// Mitsubishi GX Works2 project: 供料   PLC: FX3U/FX3UC

PROGRAM MAIN
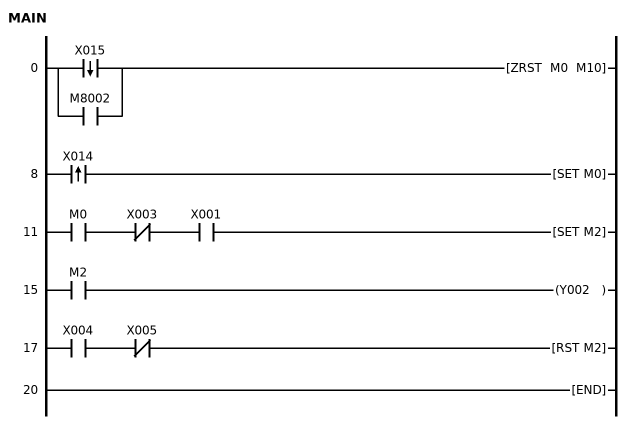
0     LDF     X015
      OR      M8002
      ZRST    M0 M10
8     LDP     X014
      SET     M0
11    LD      M0
      ANI     X003
      AND     X001
      SET     M2
15    LD      M2
      OUT     Y002
17    LD      X004
      ANI     X005
      RST     M2
20    END
END_PROGRAM
